// SIMATIC S7-200 project (STEP 7-Micro/WIN), CPU 224 UN REL 02.02

SYMBOL_TABLE USER1
sensor1          I0.0
sensor2          I0.1
sensor3          I0.2
sensor4          I0.3
sensor5          I0.4
sensor6          I0.5
sensor7          I0.6
con1             Q0.2
con2             Q0.0
con3             Q0.7
Red              Q1.2
Green            Q1.3
Yellow           Q1.4
Rod              Q0.3
TN1              Q0.4
Suc              Q0.5
Cy1              Q0.6
Cy2              Q0.1
Grip             Q1.0
TN2              Q1.1
C1S1             I0.7
C1S2             I1.0
C2S1             I1.1
C2S2             I1.2
END_SYMBOL_TABLE

ORGANIZATION_BLOCK MAIN:OB1
TITLE=PROGRAM COMMENTS
BEGIN
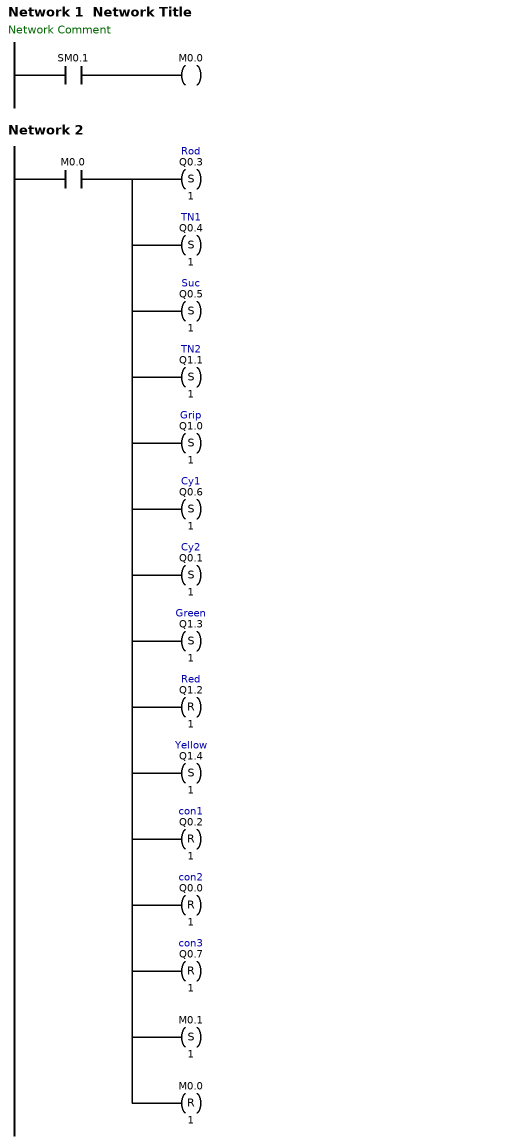
Network 1 // Network Title
// Network Comment
LD     SM0.1
=      M0.0
Network 2
LD     M0.0
S      Rod:Q0.3, 1
S      TN1:Q0.4, 1
S      Suc:Q0.5, 1
S      TN2:Q1.1, 1
S      Grip:Q1.0, 1
S      Cy1:Q0.6, 1
S      Cy2:Q0.1, 1
S      Green:Q1.3, 1
R      Red:Q1.2, 1
S      Yellow:Q1.4, 1
R      con1:Q0.2, 1
R      con2:Q0.0, 1
R      con3:Q0.7, 1
S      M0.1, 1
R      M0.0, 1
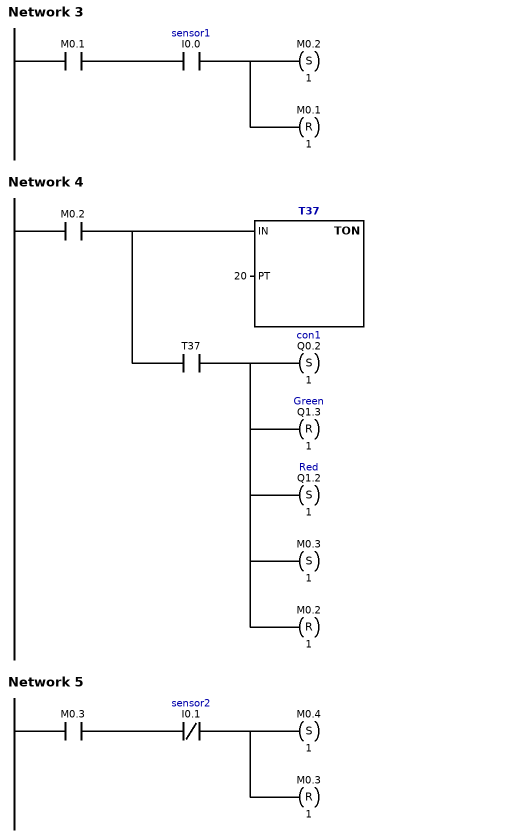
Network 3
LD     M0.1
A      sensor1:I0.0
S      M0.2, 1
R      M0.1, 1
Network 4
LD     M0.2
TON    T37, 20
A      T37
S      con1:Q0.2, 1
R      Green:Q1.3, 1
S      Red:Q1.2, 1
S      M0.3, 1
R      M0.2, 1
Network 5
LD     M0.3
AN     sensor2:I0.1
S      M0.4, 1
R      M0.3, 1
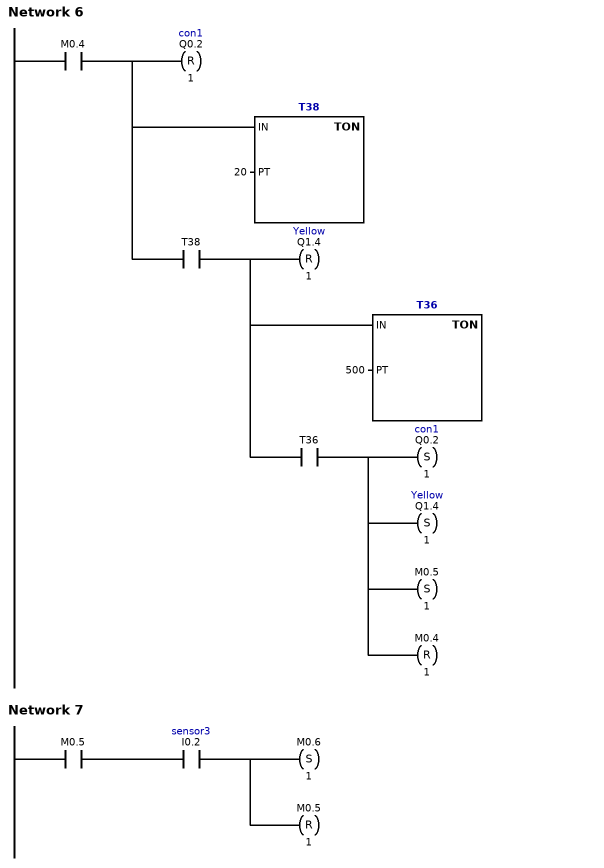
Network 6
LD     M0.4
R      con1:Q0.2, 1
TON    T38, 20
A      T38
R      Yellow:Q1.4, 1
TON    T36, 500
A      T36
S      con1:Q0.2, 1
S      Yellow:Q1.4, 1
S      M0.5, 1
R      M0.4, 1
Network 7
LD     M0.5
A      sensor3:I0.2
S      M0.6, 1
R      M0.5, 1
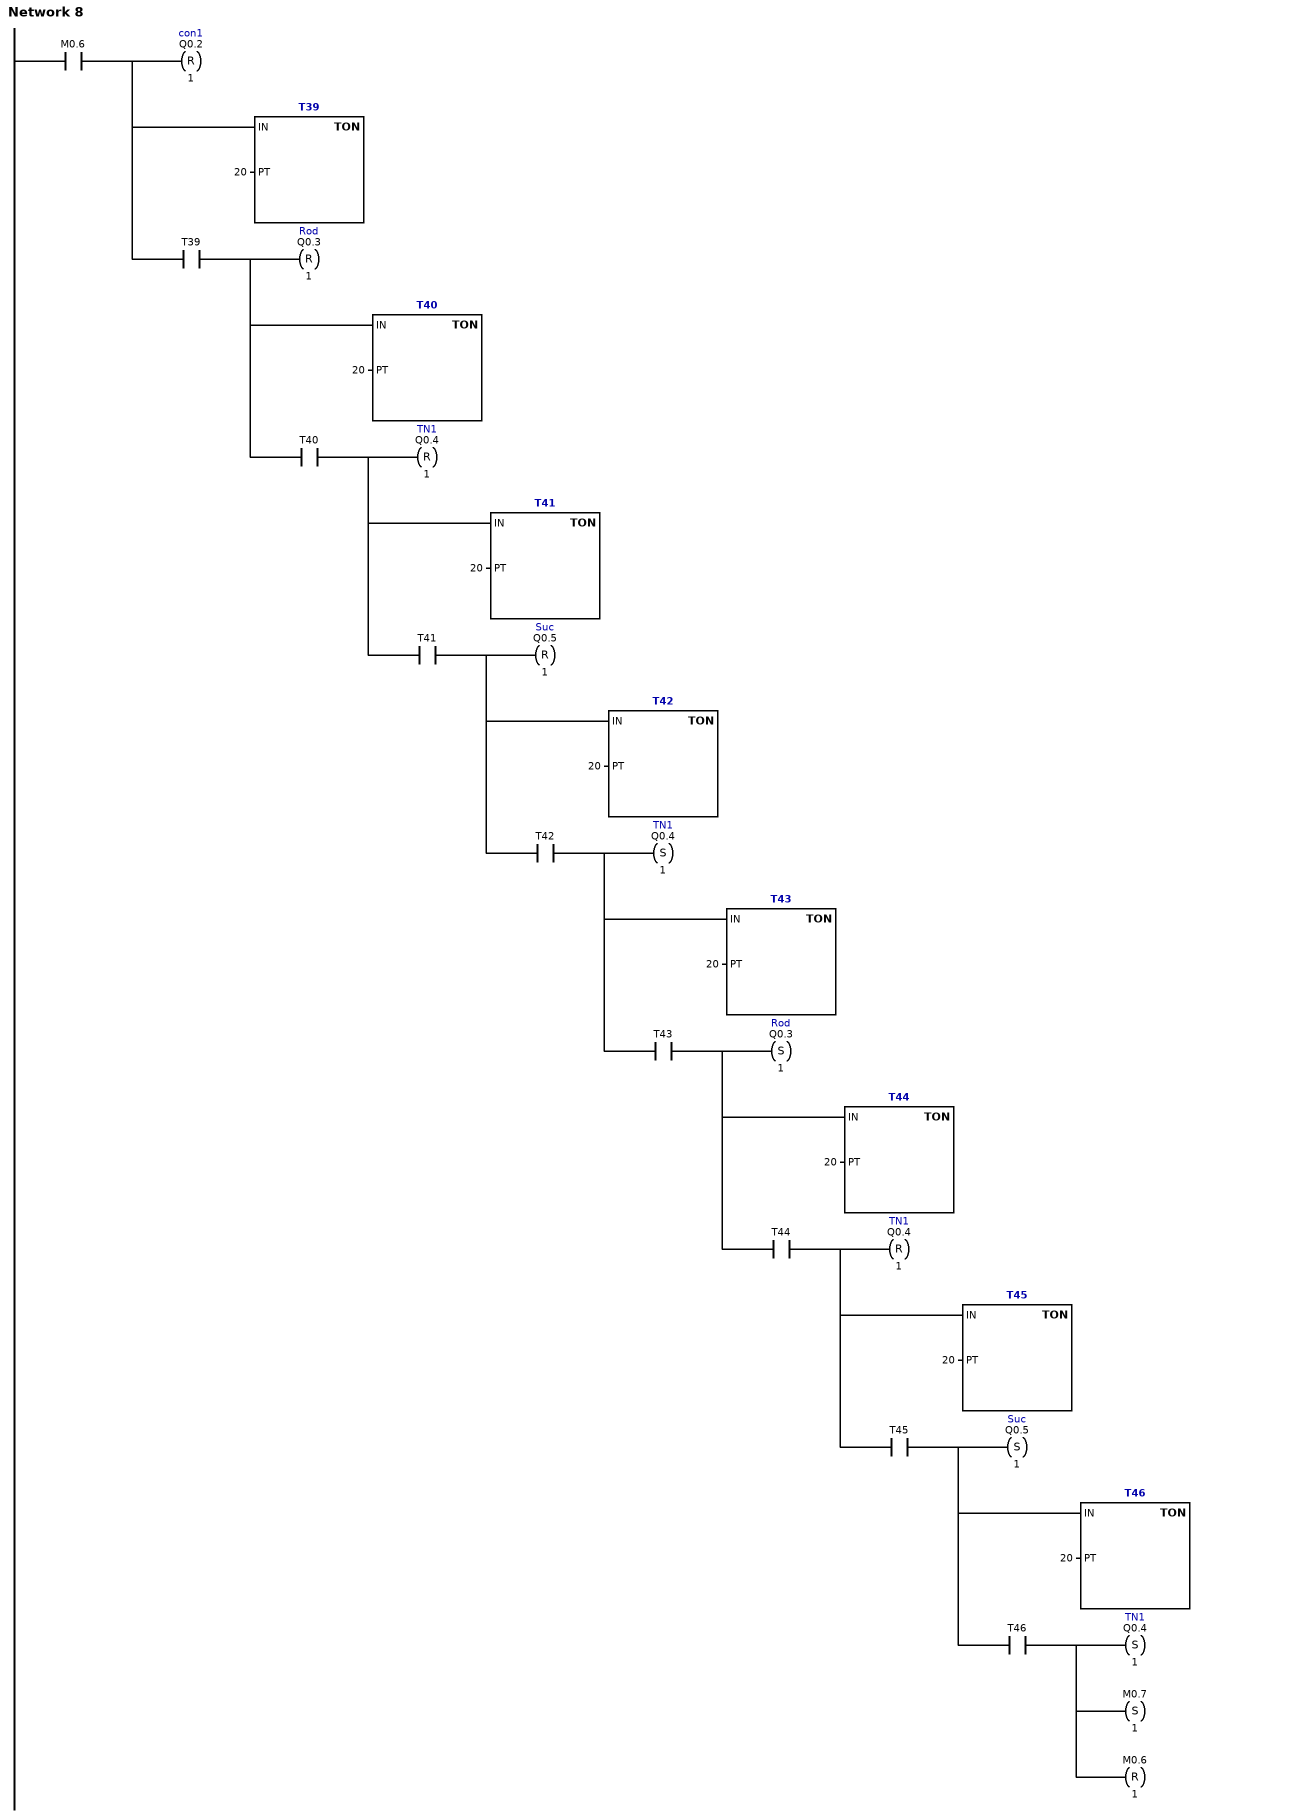
Network 8
LD     M0.6
R      con1:Q0.2, 1
TON    T39, 20
A      T39
R      Rod:Q0.3, 1
TON    T40, 20
A      T40
R      TN1:Q0.4, 1
TON    T41, 20
A      T41
R      Suc:Q0.5, 1
TON    T42, 20
A      T42
S      TN1:Q0.4, 1
TON    T43, 20
A      T43
S      Rod:Q0.3, 1
TON    T44, 20
A      T44
R      TN1:Q0.4, 1
TON    T45, 20
A      T45
S      Suc:Q0.5, 1
TON    T46, 20
A      T46
S      TN1:Q0.4, 1
S      M0.7, 1
R      M0.6, 1
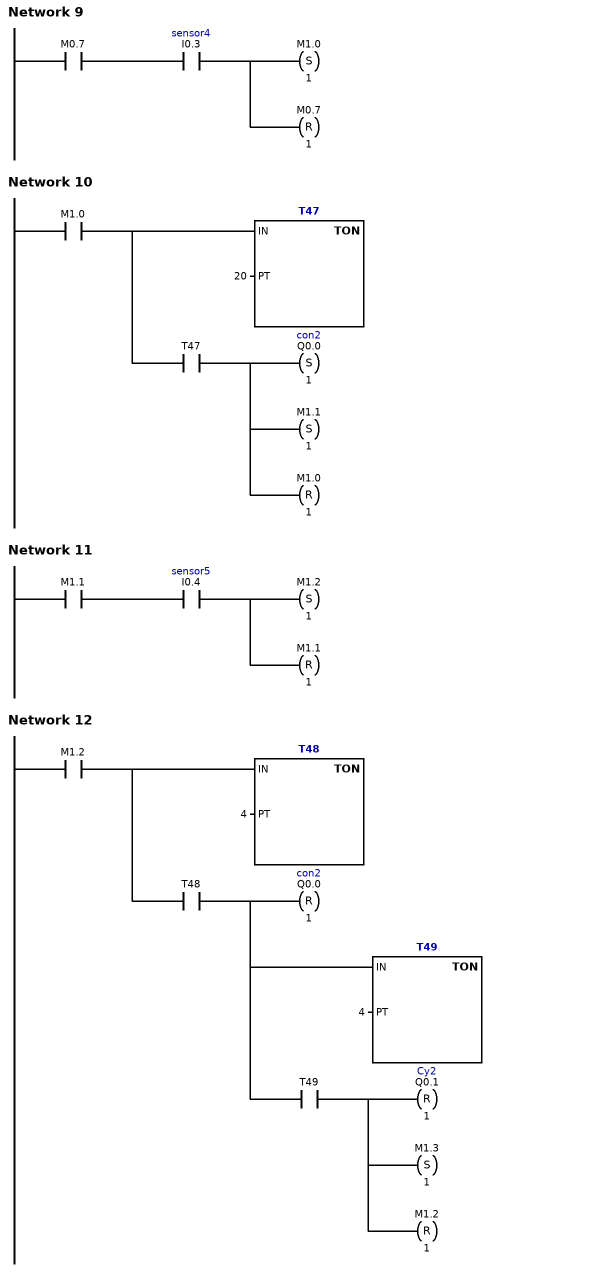
Network 9
LD     M0.7
A      sensor4:I0.3
S      M1.0, 1
R      M0.7, 1
Network 10
// (network saved uncompiled; LAD cells follow)
// row 0: c0 -| |- M1.0 v  c1 --  c2 [TON T47 IN:=power@row0, PT:=20]
// row 1: c0 ^v  c2 [box]
// row 2: c0 ^  c1 -| |- T47 v  c2 -(S) con2:Q0.0, 1
// row 3: c1 ^v  c2 -(S) M1.1, 1
// row 4: c1 ^  c2 -(R) M1.0, 1
Network 11
LD     M1.1
A      sensor5:I0.4
S      M1.2, 1
R      M1.1, 1
Network 12
LD     M1.2
TON    T48, 4
A      T48
R      con2:Q0.0, 1
TON    T49, 4
A      T49
R      Cy2:Q0.1, 1
S      M1.3, 1
R      M1.2, 1
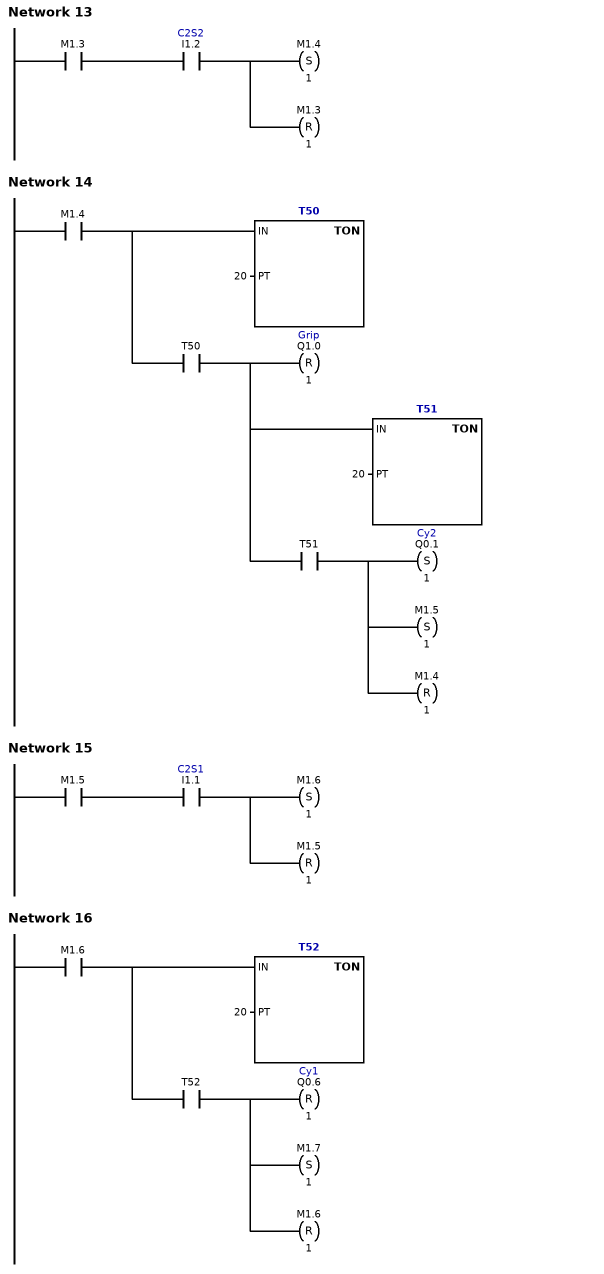
Network 13
LD     M1.3
A      C2S2:I1.2
S      M1.4, 1
R      M1.3, 1
Network 14
LD     M1.4
TON    T50, 20
A      T50
R      Grip:Q1.0, 1
TON    T51, 20
A      T51
S      Cy2:Q0.1, 1
S      M1.5, 1
R      M1.4, 1
Network 15
LD     M1.5
A      C2S1:I1.1
S      M1.6, 1
R      M1.5, 1
Network 16
LD     M1.6
TON    T52, 20
A      T52
R      Cy1:Q0.6, 1
S      M1.7, 1
R      M1.6, 1
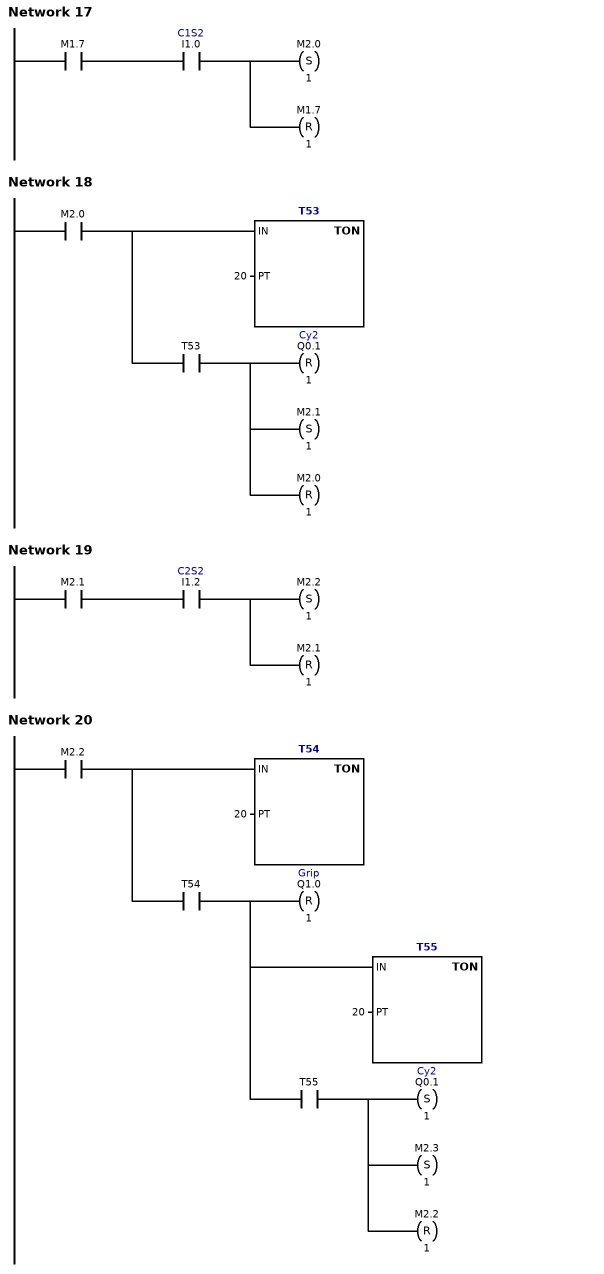
Network 17
LD     M1.7
A      C1S2:I1.0
S      M2.0, 1
R      M1.7, 1
Network 18
LD     M2.0
TON    T53, 20
A      T53
R      Cy2:Q0.1, 1
S      M2.1, 1
R      M2.0, 1
Network 19
LD     M2.1
A      C2S2:I1.2
S      M2.2, 1
R      M2.1, 1
Network 20
LD     M2.2
TON    T54, 20
A      T54
R      Grip:Q1.0, 1
TON    T55, 20
A      T55
S      Cy2:Q0.1, 1
S      M2.3, 1
R      M2.2, 1
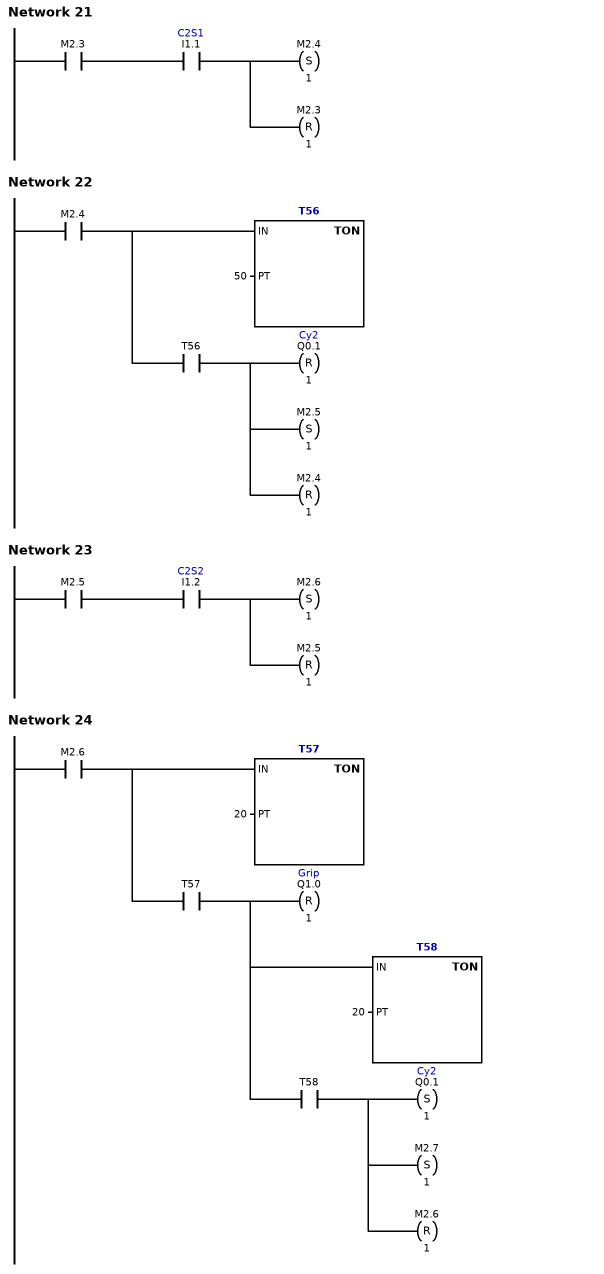
Network 21
LD     M2.3
A      C2S1:I1.1
S      M2.4, 1
R      M2.3, 1
Network 22
LD     M2.4
TON    T56, 50
A      T56
R      Cy2:Q0.1, 1
S      M2.5, 1
R      M2.4, 1
Network 23
LD     M2.5
A      C2S2:I1.2
S      M2.6, 1
R      M2.5, 1
Network 24
LD     M2.6
TON    T57, 20
A      T57
R      Grip:Q1.0, 1
TON    T58, 20
A      T58
S      Cy2:Q0.1, 1
S      M2.7, 1
R      M2.6, 1
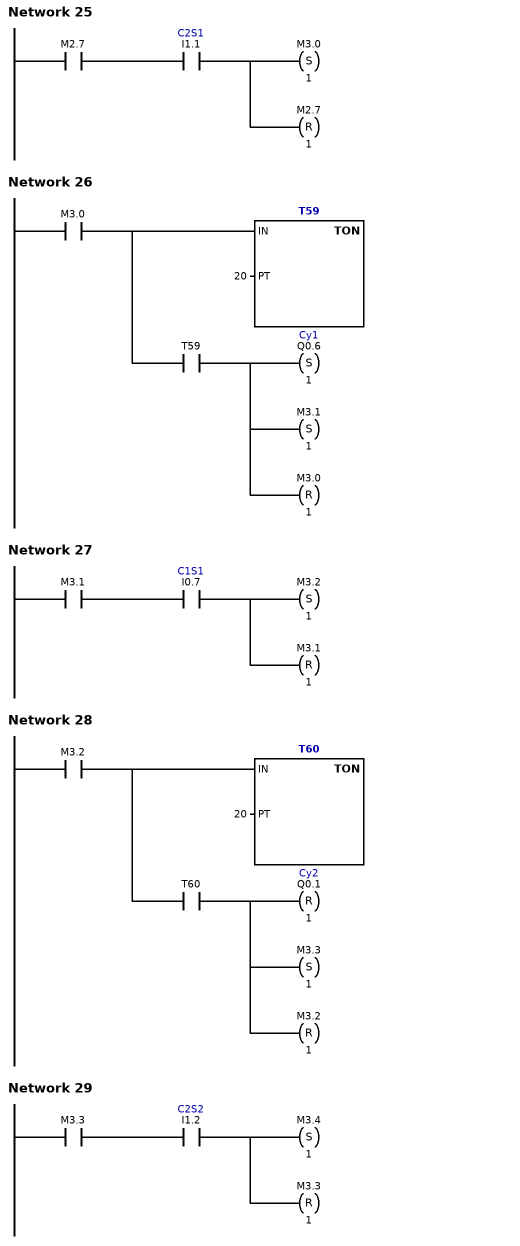
Network 25
LD     M2.7
A      C2S1:I1.1
S      M3.0, 1
R      M2.7, 1
Network 26
LD     M3.0
TON    T59, 20
A      T59
S      Cy1:Q0.6, 1
S      M3.1, 1
R      M3.0, 1
Network 27
LD     M3.1
A      C1S1:I0.7
S      M3.2, 1
R      M3.1, 1
Network 28
LD     M3.2
TON    T60, 20
A      T60
R      Cy2:Q0.1, 1
S      M3.3, 1
R      M3.2, 1
Network 29
LD     M3.3
A      C2S2:I1.2
S      M3.4, 1
R      M3.3, 1
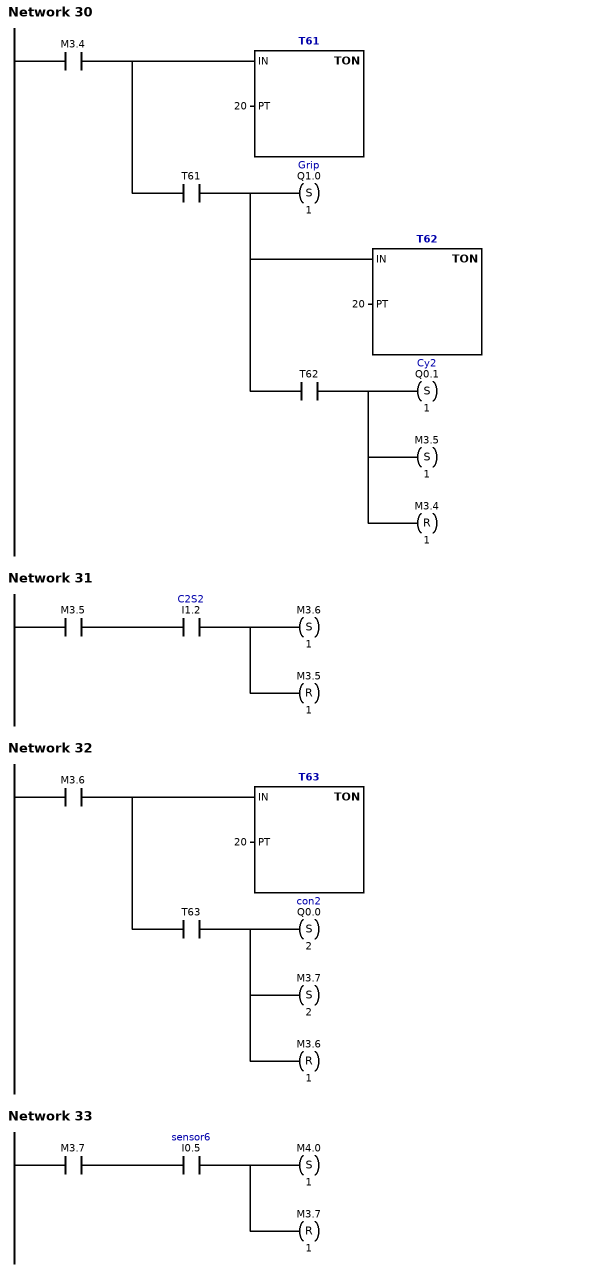
Network 30
LD     M3.4
TON    T61, 20
A      T61
S      Grip:Q1.0, 1
TON    T62, 20
A      T62
S      Cy2:Q0.1, 1
S      M3.5, 1
R      M3.4, 1
Network 31
LD     M3.5
A      C2S2:I1.2
S      M3.6, 1
R      M3.5, 1
Network 32
LD     M3.6
TON    T63, 20
A      T63
S      con2:Q0.0, 2
S      M3.7, 2
R      M3.6, 1
Network 33
LD     M3.7
A      sensor6:I0.5
S      M4.0, 1
R      M3.7, 1
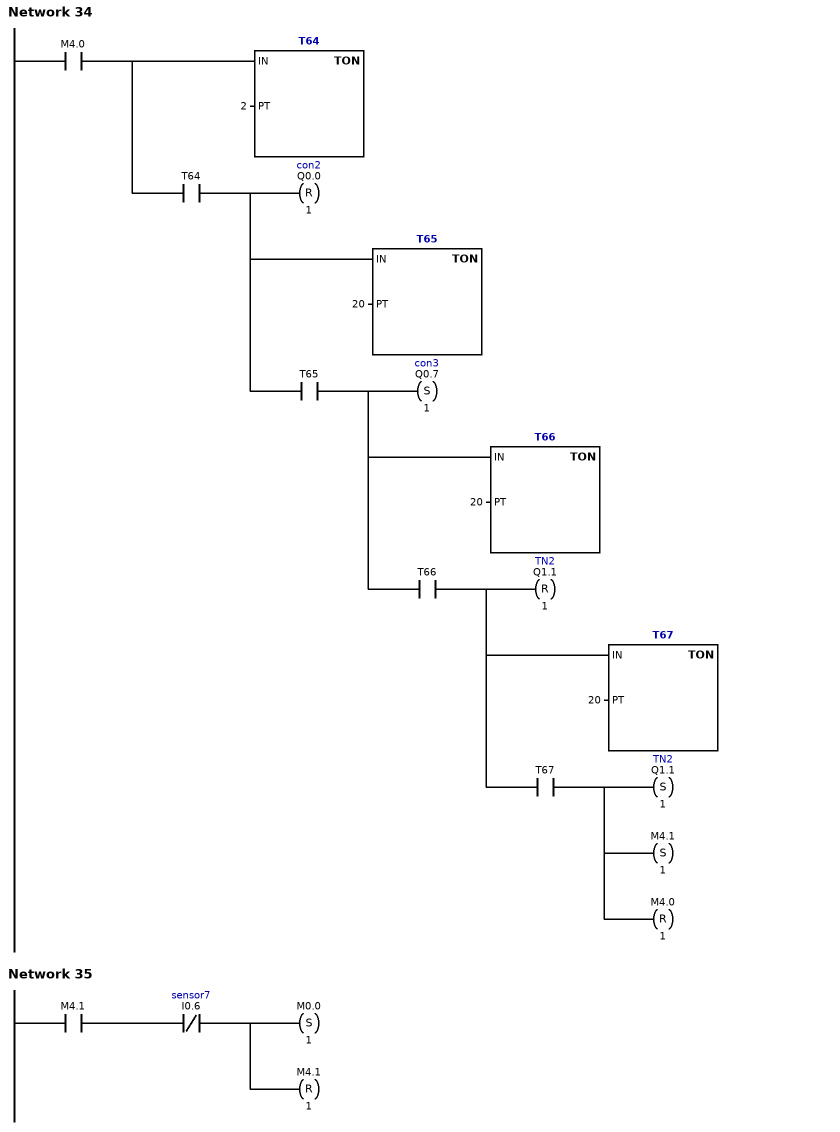
Network 34
LD     M4.0
TON    T64, 2
A      T64
R      con2:Q0.0, 1
TON    T65, 20
A      T65
S      con3:Q0.7, 1
TON    T66, 20
A      T66
R      TN2:Q1.1, 1
TON    T67, 20
A      T67
S      TN2:Q1.1, 1
S      M4.1, 1
R      M4.0, 1
Network 35
LD     M4.1
AN     sensor7:I0.6
S      M0.0, 1
R      M4.1, 1
END_ORGANIZATION_BLOCK
